FUNCTION Convert_LWORD_TO_DT : Hresult
VAR_INPUT
	in : LWORD;
	out : REFERENCE TO DT;
END_VAR
VAR
	converted : DT;
END_VAR
VAR CONSTANT
	INCOMPATIBLE : HRESULT := 16#9811070E;
END_VAR

converted := LWORD_TO_DT(in);

IF (DT_TO_LWORD(converted) <> in) THEN
	Convert_LWORD_TO_DT := INCOMPATIBLE;
	RETURN;
END_IF

out := converted;

END_FUNCTION

(* stored: Version 1.1.0.1, ProductVersion 3.1.4024.12
   POU Convert_LWORD_TO_DT: Id {ea2d0f46-694e-44aa-8264-0d90aa086157}, SpecialFunc None *)
